// TIA Portal project "Ejercicio1" (V15.1)

(* hardware
DEVICE "S7-1200 station_2"  S7-1200 Station
   slot 0: "Rack_0"  S7-1200 Rack  Rack  V1.0
   slot 1: "PLC_0"  CPU 1215C AC/DC/Rly  6ES7 215-1BG40-0XB0  V4.2
DEVICE "HMI_1"  KTP700 Basic PN
   slot 0: "HMI_1"  KTP700 Basic PN  6AV2 123-2GB03-0AX0  15.1.0.0
   slot 1: "HMI_RT_1"  KTP700 Basic PN  6AV2 123-2GB03-0AX0  15.1.0.0
   slot 5: "HMI_1.IE_CP_1"  PROFINET Interface  15.0.1.0
      slot 1: "Interfaz PROFINET_1"  PROFINET Interface
         slot 1: "Port_1"  Port
*)

// ===== PLC "PLC_0"  CPU 1215C AC/DC/Rly =====

VAR_GLOBAL   // PLC tag table "Tabla de variables estándar"
   "Interruptor ON/OFF" AT %M0.0 : Bool;
   "Palanca de giro positivo motor" AT %M0.1 : Bool;
   "Palanca de giro negativo motor" AT %M0.2 : Bool;
   "Lampara funcionamiento" AT %M10.0 : Bool;
   "Lampara sentido de positivo giro" AT %M10.1 : Bool;
   "Lampara sentido negativo de giro" AT %M10.2 : Bool;
   "Contactor giro positivo motor" AT %M10.3 : Bool;
   "Contactor giro negativo motor" AT %M10.4 : Bool;
   "Sensor de temperatura" AT %M0.3 : Bool;
   "Piloto panel de mando" AT %M10.5 : Bool;
END_VAR

ORGANIZATION_BLOCK "Main"   // OB1, LAD, ProgramCycle
TITLE = "Main Program Sweep (Cycle)"
{ S7_Optimized_Access := 'TRUE' }
VERSION : 0.1
   VAR_INPUT
      Initial_Call : Bool;   // Initial call of this OB
      Remanence : Bool;   // =True, if remanent data are available
   END_VAR
   VAR_TEMP   // added for the SCL form of the ladder/FBD networks
      _w1 : Bool;
      _w2 : Bool;
   END_VAR
BEGIN

REGION Network 1
   // Ejercicio 1
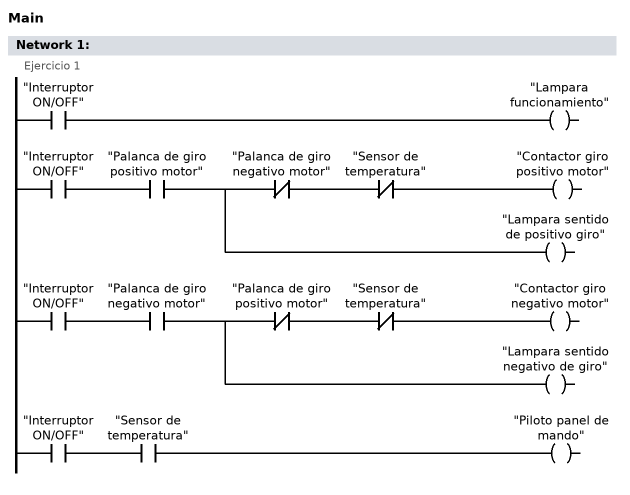
   RUNG wire#powerrail
      Contact( "Interruptor ON/OFF" )
      Coil( "Lampara funcionamiento" )
   END_RUNG
   RUNG wire#powerrail
      Contact( "Interruptor ON/OFF" )
      Contact( "Palanca de giro positivo motor" )
      wire#w1
      I_Contact( "Palanca de giro negativo motor" )
      I_Contact( "Sensor de temperatura" )
      Coil( "Contactor giro positivo motor" )
   END_RUNG
   RUNG wire#w1
      Coil( "Lampara sentido de positivo giro" )
   END_RUNG
   RUNG wire#powerrail
      Contact( "Interruptor ON/OFF" )
      Contact( "Palanca de giro negativo motor" )
      wire#w2
      I_Contact( "Palanca de giro positivo motor" )
      I_Contact( "Sensor de temperatura" )
      Coil( "Contactor giro negativo motor" )
   END_RUNG
   RUNG wire#w2
      Coil( "Lampara sentido negativo de giro" )
   END_RUNG
   RUNG wire#powerrail
      Contact( "Interruptor ON/OFF" )
      Contact( "Sensor de temperatura" )
      Coil( "Piloto panel de mando" )
   END_RUNG
   // the same network as SCL:
   "Lampara funcionamiento" := "Interruptor ON/OFF";
   #_w1 := "Interruptor ON/OFF" AND "Palanca de giro positivo motor";
   "Contactor giro positivo motor" := #_w1 AND NOT "Palanca de giro negativo motor" AND NOT "Sensor de temperatura";
   "Lampara sentido de positivo giro" := #_w1;
   #_w2 := "Interruptor ON/OFF" AND "Palanca de giro negativo motor";
   "Contactor giro negativo motor" := #_w2 AND NOT "Palanca de giro positivo motor" AND NOT "Sensor de temperatura";
   "Lampara sentido negativo de giro" := #_w2;
   "Piloto panel de mando" := "Interruptor ON/OFF" AND "Sensor de temperatura";
END_REGION
END_ORGANIZATION_BLOCK

(* ===== HMI "HMI_RT_1" =====
system functions are stored by id; their names below are inferred from use
connection "HMI_Conexión_1": ETHERNET, SMART_S7_1200_OMS

HMI tags "Tabla de variables estándar"
   "Número_imagen_variable" : UInt, internal
   "Lampara funcionamiento" : Bool = PLC "Lampara funcionamiento" AT %M10.0, 1 s
   "Lampara sentido de positivo giro" : Bool = PLC "Lampara sentido de positivo giro" AT %M10.1, 1 s
   "Lampara sentido negativo de giro" : Bool = PLC "Lampara sentido negativo de giro" AT %M10.2, 1 s
   "Piloto panel de mando" : Bool = PLC "Piloto panel de mando" AT %M10.5, 1 s
   "Interruptor ON/OFF" : Bool = PLC "Interruptor ON/OFF" AT %M0.0, 1 s
   "Palanca de giro positivo motor" : Bool = PLC "Palanca de giro positivo motor" AT %M0.1, 1 s
   "Palanca de giro negativo motor" : Bool = PLC "Palanca de giro negativo motor" AT %M0.2, 1 s

text list "Nombre_imagen_lista_texto": 1 'Imagen raíz'

Template "Plantilla_1" 800x480
   Button "Salir" at 714,429 size 71x50; TextOff 'Salir'; PictureOff "ExitRuntime_KTP700_Basic_PN_TR"; PictureOn "ExitRuntime_KTP700_Basic_PN_TR"
      on Release: StopRuntime(0)
   Button "Template_Button" at 614,429 size 71x50; TextOff 'Text'
   Button "Template_Button_1" at 514,429 size 71x50; TextOff 'Text'
   Button "Template_Button_2" at 414,429 size 71x50; TextOff 'Text'
   Button "Template_Button_3" at 314,429 size 71x50; TextOff 'Text'
   Button "Template_Button_4" at 214,429 size 71x50; TextOff 'Text'
   Button "Avisos" at 114,429 size 71x50; TextOff 'Avisos'; PictureOff "AlarmDisplay_KTP700_Basic_PN_TR"; PictureOn "AlarmDisplay_KTP700_Basic_PN_TR"
      on Release: function_ef3f5d25("Ventana de avisos_no_acusado", -1)
   Button "Imagen inicial" at 14,429 size 71x50; TextOff 'Imagen inicial'; PictureOff "NavigateHome_KTP700_Basic_PN_TR"; PictureOn "NavigateHome_KTP700_Basic_PN_TR"
      on Release: ActivateScreen("Imagen raíz", 0)
   SymbolicIOField "Imagen_campo_ES_simbólico" at 2,9 size 691x33; TextOff '0'; TextOn '1'; TextList "Nombre_imagen_lista_texto"
      ProcessValue <- "Número_imagen_variable"
      on Change: ActivateScreenByNumber("Número_imagen_variable", 0)
   DateTimeField "HmiScreenItemData" at 695,25 size 105x25
   DateTimeField "HmiScreenItemData_1" at 695,0 size 105x25

screen "Imagen raíz" 800x480, template "Plantilla_1"
   on GenerateScreen: SetTag("Número_imagen_variable", 1)
   Circle "Círculo_1" at 476,96 size 48x48
      Appearance <- "Lampara funcionamiento"
   Circle "Círculo_2" at 476,192 size 48x48
      Appearance <- "Lampara sentido de positivo giro"
   Circle "Círculo_3" at 476,259 size 48x48
      Appearance <- "Lampara sentido negativo de giro"
   Circle "Círculo_4" at 476,342 size 48x48
      Appearance <- "Piloto panel de mando"
   TextField "Campo de texto_1" at 536,110 size 192x23; Text 'LED de funcionamiento'
   TextField "Campo de texto_2" at 536,203 size 142x23; Text 'LED giro positivo'
   TextField "Campo de texto_3" at 536,271 size 149x23; Text 'LED giro negativo'
   TextField "Campo de texto_4" at 536,357 size 218x23; Text 'Piloto del panel de mando'
   Switch "Interruptor_1" at 74,101 size 64x32; CaptionText 'Switch'; TextOff 'OFF'; TextOn 'ON'
      ProcessValue <- "Interruptor ON/OFF"
   Switch "Interruptor_2" at 74,206 size 64x32; CaptionText 'Switch'; TextOff 'OFF'; TextOn 'ON'
      ProcessValue <- "Palanca de giro positivo motor"
   Switch "Interruptor_3" at 74,254 size 64x32; CaptionText 'Switch'; TextOff 'OFF'; TextOn 'ON'
      ProcessValue <- "Palanca de giro negativo motor"
   TextField "Campo de texto_5" at 149,110 size 165x23; Text 'Interruptor ON/OFF'
   TextField "Campo de texto_6" at 149,217 size 200x23; Text 'Palanca de giro positivo'
   TextField "Campo de texto_7" at 149,259 size 207x23; Text 'Palanca de giro negativo'
*)